FUNCTION_BLOCK StringBuilderExtBufferTest EXTENDS TcUnit.FB_TestSuite
VAR
END_VAR

AppendAndClear();

METHOD AppendAndClear : BOOL
VAR
	buffer : STRING(2000);
	builder : StringBuilderExtBuffer(buffer);
	
	testValue : STRING := ' very long strings';
END_VAR
TcUnit.TEST('Append and Clear');

builder
	.Clear()
	.Append('SB with external buffer')
	.Append(' is meant for')
	.AppendByPointer(ADR(testValue));

AssertEquals_STRING(
	Expected := 'SB with external buffer is meant for very long strings',
	Actual := buffer,
	Message := 'Strings should be properly appended');

builder.Clear();

AssertEquals_BOOL(
	Expected := TRUE,
	Actual := builder.IsEmpty,
	Message := 'Buffer should be empty');
	
TEST_FINISHED();
END_METHOD

END_FUNCTION_BLOCK

(* stored: Version 1.1.0.1, ProductVersion 3.1.4024.12
   POU StringBuilderExtBufferTest: Id {aff41a11-6836-079e-1b20-bff758e05ee0}, SpecialFunc None
   Method AppendAndClear: Id {4da07407-4d74-0d70-3110-4bd92ed5ae18} *)
